FUNCTION_BLOCK InfluentFeedLogic (* CAT Function Block Type *)
  (* Standard: 61499-2 *)
  (* Version 0.0, 15/09/2026, template *)
  PACKAGE Hidryco.HidrycoLib;
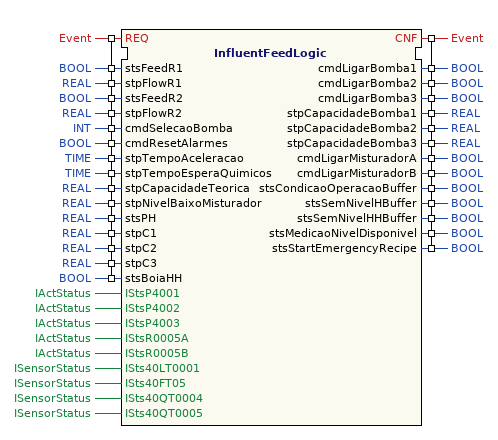
  EVENT_INPUT
    REQ WITH stsFeedR1, stpFlowR1, stsFeedR2, stpFlowR2, cmdSelecaoBomba, cmdResetAlarmes, stpTempoAceleracao, stpTempoEsperaQuimicos, stpCapacidadeTeorica, stpNivelBaixoMisturador, stsPH, stpC1, stpC2, stpC3, stsBoiaHH;
  END_EVENT
  EVENT_OUTPUT
    CNF WITH cmdLigarBomba1, cmdLigarBomba2, cmdLigarBomba3, stpCapacidadeBomba1, stpCapacidadeBomba2, stpCapacidadeBomba3, cmdLigarMisturadorA, cmdLigarMisturadorB, stsCondicaoOperacaoBuffer, stsSemNivelHBuffer, stsSemNivelHHBuffer, stsMedicaoNivelDisponivel, stsStartEmergencyRecipe;
  END_EVENT
  VAR_INPUT
    stsFeedR1 : BOOL;
    stpFlowR1 : REAL;
    stsFeedR2 : BOOL;
    stpFlowR2 : REAL;
    cmdSelecaoBomba : INT;
    cmdResetAlarmes : BOOL;
    stpTempoAceleracao : TIME; (* Espera antes de controlar as duas bombas juntas *)
    stpTempoEsperaQuimicos : TIME; (* Espera para reiniciar após pH e condutividade normalizarem *)
    stpCapacidadeTeorica : REAL; (* Vazão nominal, para a malha aberta *)
    stpNivelBaixoMisturador : REAL; (* Bloqueio para misturadores *)
    stsPH : REAL;
    stpC1 : REAL;
    stpC2 : REAL;
    stpC3 : REAL;
    stsBoiaHH : BOOL;
  END_VAR
  VAR_OUTPUT
    cmdLigarBomba1 : BOOL;
    cmdLigarBomba2 : BOOL;
    cmdLigarBomba3 : BOOL;
    stpCapacidadeBomba1 : REAL;
    stpCapacidadeBomba2 : REAL;
    stpCapacidadeBomba3 : REAL;
    cmdLigarMisturadorA : BOOL;
    cmdLigarMisturadorB : BOOL;
    stsCondicaoOperacaoBuffer : BOOL; (* Operating condition da fase Feed, nos dois reatores. FALSE quando o buffer não pode alimentar *)
    stsSemNivelHBuffer : BOOL;
    stsSemNivelHHBuffer : BOOL;
    stsMedicaoNivelDisponivel : BOOL;
    stsStartEmergencyRecipe : BOOL;
  END_VAR
  SOCKETS
    IStsP4001 : IActStatus;
    IStsP4002 : IActStatus;
    IStsP4003 : IActStatus;
    IStsR0005A : IActStatus;
    IStsR0005B : IActStatus;
    ISts40LT0001 : ISensorStatus;
    ISts40FT05 : ISensorStatus;
    ISts40QT0004 : ISensorStatus;
    ISts40QT0005 : ISensorStatus;
  END_SOCKETS
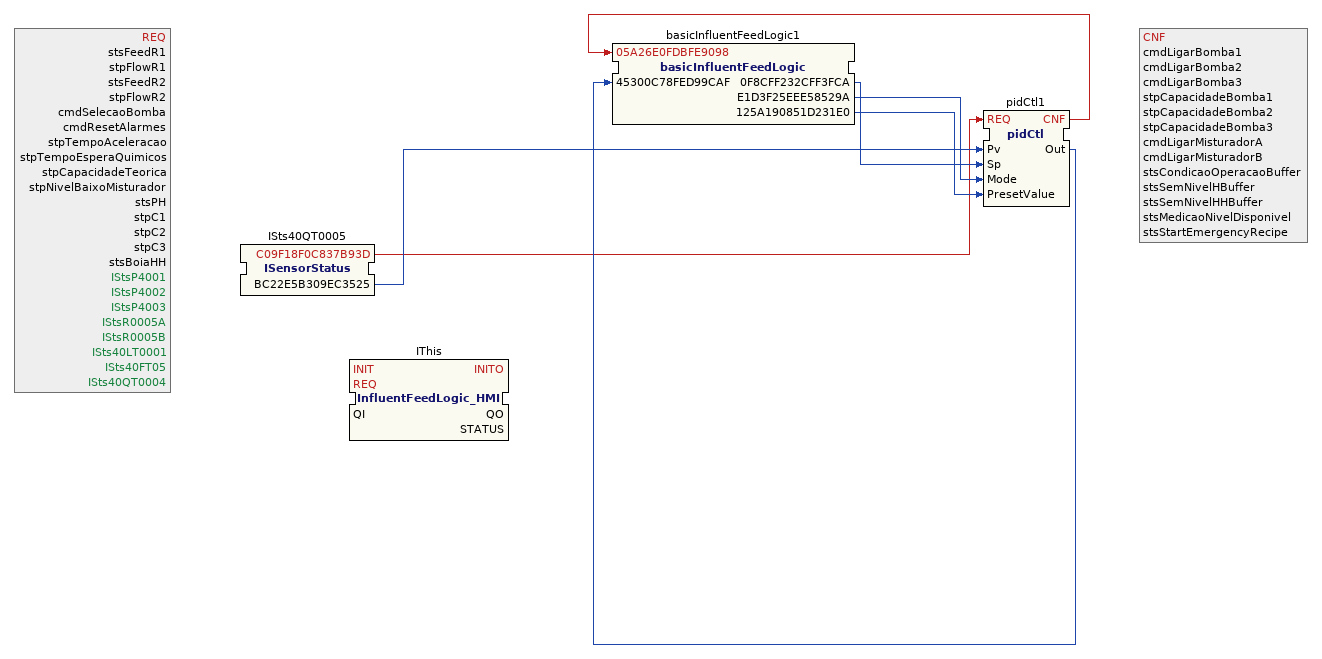
  FBS
    basicInfluentFeedLogic1 : basicInfluentFeedLogic;
    IThis : InfluentFeedLogic_HMI;
    pidCtl1 : pidCtl;
  END_FBS
  EVENT_CONNECTIONS
    ISts40QT0005.C09F18F0C837B93D TO pidCtl1.REQ;
    pidCtl1.CNF TO basicInfluentFeedLogic1.05A26E0FDBFE9098;
  END_CONNECTIONS
  DATA_CONNECTIONS
    ISts40QT0005.BC22E5B309EC3525 TO pidCtl1.Pv;
    basicInfluentFeedLogic1.0F8CFF232CFF3FCA TO pidCtl1.Sp;
    basicInfluentFeedLogic1.E1D3F25EEE58529A TO pidCtl1.Mode;
    basicInfluentFeedLogic1.125A190851D231E0 TO pidCtl1.PresetValue;
    pidCtl1.Out TO basicInfluentFeedLogic1.45300C78FED99CAF;
  END_CONNECTIONS
END_FUNCTION_BLOCK
